Yaskawa INFORM job: TEST1.JBI

/JOB
//NAME TEST1
//POS
///NPOS 5,0,5,0,0,0
///TOOL 0
///POSTYPE PULSE
///PULSE
C00000=-8101,-25260,-100961,85462,13502,-22784
C00001=-8101,-25260,-100961,85462,13502,-22784
C00002=0,0,0,0,0,0
C00003=10189,39782,-61789,107251,-41127,-20238
C00004=0,0,0,0,0,0
EC00000=184320
EC00001=0
EC00002=0
EC00003=0
EC00004=0
//INST
///DATE 2023/04/23 14:49
///ATTR SC,RW
///GROUP1 RB1,ST1
NOP
MOVJ C00000 EC00000 VJ=10.00
MOVJ C00001 EC00001 VJ=10.00
MOVJ C00002 EC00002 VJ=10.00
MOVJ C00003 EC00003 VJ=10.00
MOVJ C00004 EC00004 VJ=10.00
END
